PROGRAM MAIN
VAR
END_VAR

END_PROGRAM

(* stored: Version 1.1.0.1
   POU MAIN: Id {f1a33ef1-91ed-4177-af7d-9142b8f1473d} *)
